// TIA Portal V20 export
// export: Created 2025-12-01T14:57:43.40006Z, ExportSetting None, DisplayName Totally Integrated Automation Portal, DisplayVersion V20 Update 3, DisplayName TIA Portal Openness, DisplayVersion V20 Update 3, DisplayName TIA Portal Version Control Interface, DisplayVersion V20 Update 3, DisplayName STEP 7 Professional, DisplayVersion V20 Update 3, DisplayName STEP 7 Safety, DisplayVersion V20 Update 2, DisplayName WinCC Basic/Comfort/Advanced, DisplayVersion V20 Update 3, DisplayName WinCC Professional, DisplayVersion V20 Update 3, DisplayName WinCC Unified, DisplayVersion V20 Update 3
FUNCTION "FC501_Etiq_Router_DEMO3D" : Void   // FC501, LAD
{ S7_Optimized_Access := 'FALSE' }
// stored: AutoNumber false, SetENOAutomatically false
   VAR_INPUT
      Mesa : UInt;
   END_VAR
   VAR_OUTPUT
      Etiqueta1 : DInt;
      Etiqueta2 : DInt;
   END_VAR
   VAR_TEMP
      Digitos_Etiqueta : UInt;
      NUM_UT : DInt;
      Num_UT_2 : DInt;
      SSCC_STR : String [9];
   END_VAR
BEGIN

REGION Network 1 (SCL)
   //Función que se utiliza para poder etiquetar las unidades de carga generadas en Demo3D
   //con la etiqueta que nos manda JDT en el atributo de la UT.
   // por el tipo de datos de salida la cantidad máxima de dígitos que se pueden transformar 
   // la vamos a limitar a 9 (de 0 a 8) igual que en el router: etiqueta maxima 999999999

   #Digitos_Etiqueta := 9;

   // primero extraemos en número de UT que hay en la mesa
   #NUM_UT := "DB810_ColasMesas".Colas[#Mesa].UT_PrimeraMesa;

   IF (#NUM_UT = 0) THEN
       // si no tengo UT, relleno con cero
       #Etiqueta1 := 0;
       #Etiqueta2 := 0;

   ELSE
       Chars_TO_Strg(Chars := "DB814_UTs_Etiqueta".UT[#NUM_UT].Etiqueta,
                     pChars := 0,
                     Cnt := #Digitos_Etiqueta,
                     Strg => #SSCC_STR);

       #Etiqueta1 := STRING_TO_DINT(#SSCC_STR);

       // extraigo el dato de si hay una segunda UT en la mesa
       #Num_UT_2 := "DB812_UTs_Control".UT[#NUM_UT].UT_SiguienteMesa;

       IF (#Num_UT_2 = 0) THEN
           #Etiqueta2 := 0;
       ELSE
           Chars_TO_Strg(Chars := "DB814_UTs_Etiqueta".UT[#Num_UT_2].Etiqueta,
                         pChars := 0,
                         Cnt := #Digitos_Etiqueta,
                         Strg => #SSCC_STR);

           #Etiqueta2 := STRING_TO_DINT(#SSCC_STR);
       END_IF;

   END_IF;
END_REGION
END_FUNCTION
